// TIA Portal project "PLC_RPI_Snap7" (V17)

(* hardware
DEVICE "S71500/ET200MP-Station_1"  S7-1500 station
   slot 0: "Profilschiene_0"  6ES7 590-1***0-0AA0
   slot 1: "PLC_1"  CPU 1511-1 PN  6ES7 511-1AK00-0AB0  V1.8
   slot 2: "AI 8xU/I/RTD/TC ST_1"  AI 8xU/I/RTD/TC ST  6ES7 531-7KF00-0AB0  V2.0
   slot 3: "AI 8xU/I/RTD/TC ST_2"  AI 8xU/I/RTD/TC ST  6ES7 531-7KF00-0AB0  V2.0
   slot 4: "AI 8xU/I/RTD/TC ST_3"  AI 8xU/I/RTD/TC ST  6ES7 531-7KF00-0AB0  V2.0
   slot 5: "AI 8xU/I/RTD/TC ST_4"  AI 8xU/I/RTD/TC ST  6ES7 531-7KF00-0AB0  V2.0
   slot 6: "DI 16x24VDC BA_1"  DI 16x24VDC BA  6ES7 521-1BH10-0AA0  V1.0
*)

// ===== PLC "PLC_1"  CPU 1511-1 PN =====

VAR_GLOBAL   // PLC tag table "Standard-Variablentabelle"
   "Pusher_Sensor" AT %E0.0 : Bool;
   "Conveyor" AT %A0.0 : Bool;
   "Start" AT %E0.1 : Bool;
   "Pusher" AT %Q1.0 : Bool;
   "Pusher_+" AT %I1.0 : Bool;
   "Stop" AT %I0.2 : Bool;
   "Scan_Stop" AT %M0.0 : Bool;
   "Activate_Pusher_Timer" AT %M1.0 : Bool;
   "Tag_1" AT %M0.1 : Bool;
   "ES" AT %I0.3 : Bool;
END_VAR

DATA_BLOCK "Sorting_line"   // DB1
{ S7_Optimized_Access := 'FALSE' }
VERSION : 0.1
   VAR
      "M0.0" : Bool := false;   // HMI_Start
      "M0.1" : Bool;   // HMI_Stop
      "M0.2" : Bool;   // Box_Type
      "M1.0" : Byte;
   END_VAR
BEGIN
END_DATA_BLOCK

DATA_BLOCK "TON"   // DB2
{ S7_Optimized_Access := 'TRUE' }
VERSION : 0.1
   VAR
      TON_Start : Bool;
      TON_Time : Time;
      TON_Q : Bool;
      TON_Preset : Time := T#1S_300ms;
   END_VAR
BEGIN
END_DATA_BLOCK

// folder: System blocks/Program resources

DATA_BLOCK "Timer"   // DB3
{ S7_Optimized_Access := 'TRUE' }
AUTHOR : Simatic
FAMILY : IEC
NAME : IEC_TMR
VERSION : 1.0
// stored: InstanceOfName IEC_TIMER
"IEC_TIMER"
BEGIN
END_DATA_BLOCK

// folder: (top level)

ORGANIZATION_BLOCK "Main"   // OB1, LAD, ProgramCycle
TITLE = "Main Program Sweep (Cycle)"
{ S7_Optimized_Access := 'TRUE' }
VERSION : 0.1
   VAR_INPUT
      Initial_Call : Bool;   // Initial call of this OB
      Remanence : Bool;   // =True, if remanent data are available
   END_VAR
BEGIN

REGION Network 1
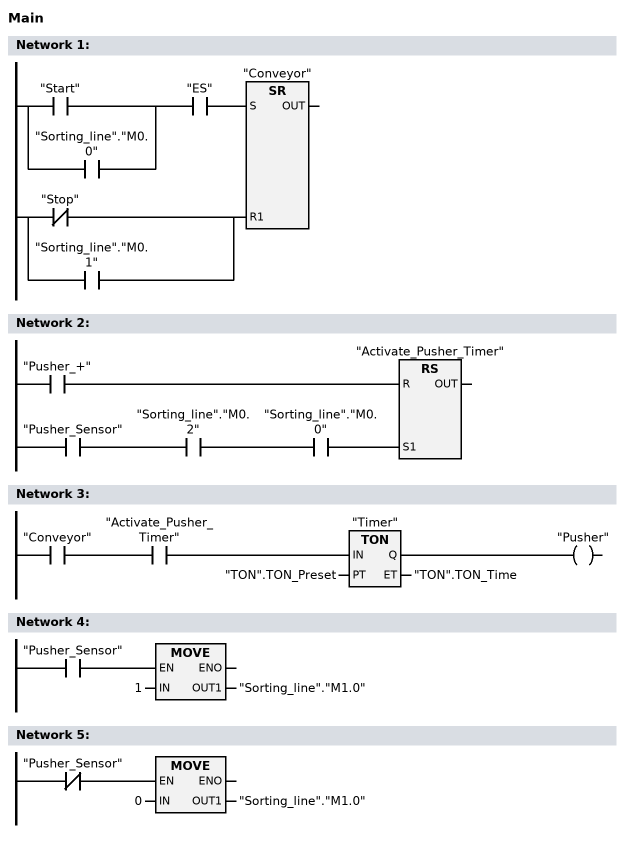
   RUNG wire#powerrail
      Contact( "Start" )
      wire#w1
      Contact( "ES" )
      S_SR(operand := "Conveyor", r1 := wire#w2)
   END_RUNG
   RUNG wire#powerrail
      Contact( "Sorting_line"."M0.0" )
   END_RUNG wire#w1
   RUNG wire#powerrail
      I_Contact( "Stop" )
   END_RUNG wire#w2
   RUNG wire#powerrail
      Contact( "Sorting_line"."M0.1" )
   END_RUNG wire#w2
   // the same network as SCL:
   IF ("Start" OR "Sorting_line"."M0.0") AND "ES" THEN
       "Conveyor" := TRUE;   // SR flip-flop
   END_IF;
   IF NOT "Stop" OR "Sorting_line"."M0.1" THEN "Conveyor" := FALSE; END_IF;
END_REGION

REGION Network 2
   RUNG wire#powerrail
      Contact( "Pusher_+" )
      S_RS(operand := "Activate_Pusher_Timer", s1 := wire#w1)
   END_RUNG
   RUNG wire#powerrail
      Contact( "Pusher_Sensor" )
      Contact( "Sorting_line"."M0.2" )
      Contact( "Sorting_line"."M0.0" )
   END_RUNG wire#w1
   // the same network as SCL:
   IF "Pusher_+" THEN
       "Activate_Pusher_Timer" := FALSE;   // RS flip-flop
   END_IF;
   IF "Pusher_Sensor" AND "Sorting_line"."M0.2" AND "Sorting_line"."M0.0" THEN
       "Activate_Pusher_Timer" := TRUE;
   END_IF;
END_REGION

REGION Network 3
   "Timer".TON(IN := "Conveyor" AND "Activate_Pusher_Timer", PT := "TON".TON_Preset, ET => "TON".TON_Time);
   "Pusher" := "Timer".Q;
END_REGION

REGION Network 4
   RUNG wire#powerrail
      Contact( "Pusher_Sensor" )
      Move(in := 1, out1 => "Sorting_line"."M1.0")
   END_RUNG
   // the same network as SCL:
   IF "Pusher_Sensor" THEN "Sorting_line"."M1.0" := 1; END_IF;
END_REGION

REGION Network 5
   RUNG wire#powerrail
      I_Contact( "Pusher_Sensor" )
      Move(in := 0, out1 => "Sorting_line"."M1.0")
   END_RUNG
   // the same network as SCL:
   IF NOT "Pusher_Sensor" THEN "Sorting_line"."M1.0" := 0; END_IF;
END_REGION
END_ORGANIZATION_BLOCK